TEXTLIST TL_TcPfw_ErrorId
  0 = 'dwTcPfwTempErrNoError'
  4098 = 'dwTcPfwTempErrBusy'
  4099 = 'dwTcPfwTempTuneErr_NoTravel'
  4100 = 'dwTcPfwTempTuneErr_NoSettling'
  4101 = 'dwTcPfwTempTuneErr_Aborted'
  4102 = 'dwTcPfwTempTuneErr_ShortOfPoints'
  4103 = 'dwTcPfwTempTuneErr_NoTop'
  4104 = ''
  4105 = 'dwTcPfwTempTuneErr_NoResponse'
  17508 = 'dwTcPfwTempErrSnsHdwFailed'
  20464 = 'dwTcPfwTempErrDisconected'
  20465 = 'dwTcPfwTempErr_NoResponse'
  20466 = 'dwTcPfwTempErrNotOperational\n'
  20467 = 'dwTcPfwTempErrIoSwapCollision\n'
  20468 = 'dwTcPfwTempErrAdsSwapCollision\n'
  20469 = 'dwTcPfwTempErrInheritedFault\n'
  20478 = 'dwTcPfwTempErrOverCurrent\n'
  20479 = 'dwTcPfwTempErrUnderCurrent'
  20480 = 'dwTcPfwTempErrSnsCommFailed'
  1800 = 'dwTcPfwTempErrBusy'
  17489 = 'dwTcPfwTempErrSnsOverrun\n'
   = ''
END_TEXTLIST

(* stored: Version 1.1.0.1, ProductVersion 3.1.4018.5
   TextList TL_TcPfw_ErrorId: Id {5fb078c8-2684-49c5-8427-63ebf416a4b0} *)
